# B&R Automation Studio project Lab2_poirts
Automation Studio 4.5.2.102

## Logical view

Binary libraries used (declarations not repeated): Runtime, Operator, AsIecCon, astime, sys_lib, asstring

### Library Logical/Libraries/DriveLib (ANSIC)

#### ConStants.var - Exported constants
```iecst
VAR CONSTANT
	CMD_SWITCHED_ON : USINT := 7;
	CMD_DISABLE_VOLTAGE : USINT := 0;
	CMD_ENABLED : USINT := 15;
	CMD_SHUTDOWN : USINT := 6;
	STATE_READY : USINT := 33;
	STATE_DISABLED : USINT := 64;
	STATE_SWITCHED_ON : USINT := 35;
	ST_INIT : USINT := 0;
	ST_UNKNOWN : USINT := 1;
	ST_OPEN : USINT := 2;
	ST_CLOSE : USINT := 3;
	ST_ACC_POS : USINT := 4;
	ST_ACC_NEG : USINT := 5;
	ST_POS : USINT := 6;
	ST_NEG : USINT := 7;
	ST_DEC_POS : USINT := 8;
	ST_DEC_NEG : USINT := 9;
END_VAR
```

#### DriveLib.fun - Exported functions and function blocks
```iecst
{REDUND_ERROR} FUNCTION_BLOCK DriveStateMachine (*TODO: Add your comment here*) (*$GROUP=User,$CAT=User,$GROUPICON=User.png,$CATICON=User.png*)
	VAR_INPUT
		state : UINT;
		enable : BOOL;
		speed : INT;
	END_VAR
	VAR_OUTPUT
		command : UINT;
	END_VAR
END_FUNCTION_BLOCK

{REDUND_ERROR} FUNCTION_BLOCK DoorStateMachine (*TODO: Add your comment here*) (*$GROUP=User,$CAT=User,$GROUPICON=User.png,$CATICON=User.png*)
	VAR_INPUT
		sw1 : {REDUND_UNREPLICABLE} BOOL;
		sw2 : {REDUND_UNREPLICABLE} BOOL;
		sw3 : {REDUND_UNREPLICABLE} BOOL;
		sw4 : {REDUND_UNREPLICABLE} BOOL;
		direction : {REDUND_UNREPLICABLE} BOOL;
	END_VAR
	VAR_OUTPUT
		speed : {REDUND_UNREPLICABLE} INT;
		state : UINT;
	END_VAR
	VAR
		osw1 : BOOL;
		osw2 : BOOL;
		osw3 : BOOL;
		osw4 : BOOL;
	END_VAR
END_FUNCTION_BLOCK

{REDUND_ERROR} FUNCTION_BLOCK LedStateMachine (*TODO: Add your comment here*) (*$GROUP=User,$CAT=User,$GROUPICON=User.png,$CATICON=User.png*)
	VAR_INPUT
		state : {REDUND_UNREPLICABLE} UINT;
	END_VAR
	VAR_OUTPUT
		led1 : {REDUND_UNREPLICABLE} BOOL;
		led2 : {REDUND_UNREPLICABLE} BOOL;
		led3 : {REDUND_UNREPLICABLE} BOOL;
		led4 : {REDUND_UNREPLICABLE} BOOL;
		timer : {REDUND_UNREPLICABLE} INT := 1;
	END_VAR
END_FUNCTION_BLOCK
```

#### DriveStateMachine.c
```c
#include <bur/plctypes.h>
#ifdef __cplusplus
	extern "C"
	{
#endif
	#include "DriveLib.h"
#ifdef __cplusplus
	};
#endif
/* TODO: Add your comment here */
void DriveStateMachine(struct DriveStateMachine* inst)
{
	UINT mask = inst->state & 0x6f;
	if(!inst->enable)
	{
		inst->command = CMD_SHUTDOWN;
	}
	else
	{
		switch (mask)
		{
			case STATE_DISABLED:
				inst->command = CMD_SHUTDOWN;
				break;

			case STATE_READY:
				inst->command = CMD_ENABLED;
				break;

			case STATE_SWITCHED_ON:
				inst->command = CMD_SWITCHED_ON;
				break;
		}
	}
}
```

#### DoorStateMachine.c
```c
#include <bur/plctypes.h>
#ifdef __cplusplus
	extern "C"
	{
#endif
	#include "DriveLib.h"
#ifdef __cplusplus
	};
#endif
/* TODO: Add your comment here */
void DoorStateMachine(struct DoorStateMachine* inst)
{
	inst->direction=!inst->direction;

	//State init
	/*if(inst->sw1==0 && inst->sw2==0 && inst->sw3==0 && inst->sw4==0)
	{
		inst->state = ST_INIT;
	}
	if(inst->state == ST_INIT)
	{

		inst->state = ST_UNKNOWN;
	}
	//state unknown
	if(inst->state == ST_UNKNOWN)
	{
		inst->state = ST_CLOSE ;
	}*/

	//открытие двери
	if(/*inst->state == ST_CLOSE &&*/ inst->sw1 != inst->osw1 && inst->direction==0)
	{
		inst->state = ST_ACC_POS ;
		inst->speed = -200;
	}

	if(/*inst->state == ST_ACC_POS &&*/ inst->sw2 != inst->osw2 && inst->direction == 0)
	{
		inst->state = ST_POS ;
		inst->speed = -600;
	}

	if(/*inst->state == ST_POS  &&*/ inst->sw3 != inst->osw3 && inst->direction == 0)
	{
		inst->state = ST_DEC_POS;
		inst->speed = -200;
	}

	if(/*inst->state == ST_DEC_POS &&*/ inst->sw4 != inst->osw4 && inst->direction == 0)
	{
		inst->state = ST_OPEN;
		inst->speed = 0;
	}

	//закрытие двери
	if(/*inst->state == ST_OPEN &&*/ inst->sw4 != inst->osw4 && inst->direction==1)
	{
		inst->state = ST_ACC_NEG;
		inst->speed = 200;
	}

	if(/*inst->state == ST_ACC_NEG &&*/ inst->sw3 != inst->osw3 && inst->direction == 1)
	{
		inst->state = ST_NEG;
		inst->speed = 600;
	}

	if(/*inst->state == ST_NEG &&*/ inst->sw2 != inst->osw2 && inst->direction == 1)
	{
		inst->state = ST_DEC_NEG;
		inst->speed = 200;
	}

	if(/*inst->state == ST_DEC_NEG &&*/ inst->sw1 != inst->osw1 && inst->direction == 1)
	{
		inst->state = ST_CLOSE;
		inst->speed = 0;
	}
	inst->osw1 = inst->sw1;
	inst->osw2 = inst->sw2;
	inst->osw3 = inst->sw3;
	inst->osw4 = inst->sw4;

}
```

#### LedStateMachine.c
```c
#include <bur/plctypes.h>
#ifdef __cplusplus
	extern "C"
	{
#endif
	#include "DriveLib.h"
#ifdef __cplusplus
	};
#endif
/* TODO: Add your comment here */
void LedStateMachine(struct LedStateMachine* inst)
{

	if(inst->state == ST_ACC_POS)
	{
		inst->led1 = 0;
		if(inst->timer == 3 )
		{
			inst->led2 = !inst->led2;
		}
		inst->led3 = 1;
		inst->led4 = 1;
	}

	if(inst->state == ST_POS)
	{
		inst->led1 = 0;
		inst->led2 = 0;
		inst->led3 = !inst->led3;
		inst->led4 = 1;
	}

	if(inst->state == ST_DEC_POS)
	{

		inst->led1 = 0;
		inst->led2 = 0;
		inst->led3 = 0;
		if(inst->timer == 3 )
		{
			inst->led4 = !inst->led4;
		}
	}

	if(inst->state == ST_OPEN)
	{
		inst->led1 = 0;
		inst->led2 = 0;
		inst->led3 = 0;
		inst->led4 = 0;
	}

	//закрытие двери
	if(inst->state == ST_ACC_NEG )
	{
		inst->led1 = 0;
		inst->led2 = 0;
		if(inst->timer == 3 )
		{
			inst->led3 = !inst->led3;
		}
		inst->led4 = 1;
	}

	if(inst->state == ST_NEG)
	{
		inst->led1 = 0;
		inst->led2 =!inst->led2;
		inst->led3 = 1;
		inst->led4 = 1;
	}

	if(inst->state == ST_DEC_NEG )
	{
		if(inst->timer == 3 )
		{
			inst->led1 = !inst->led1;
		}
		inst->led2 = 1;
		inst->led3 = 1;
		inst->led4 = 1;
	}

	if(inst->state == ST_CLOSE)
	{
		inst->led1 = 1;
		inst->led2 = 1;
		inst->led3 = 1;
		inst->led4 = 1;
	}

	if(inst->timer == 3)
		inst->timer = 0;

	inst->timer++;
}
```

### Program Logical/Program (ANSIC)

#### Init.c - Initialization code
```c
#include <bur/plctypes.h>

#ifdef _DEFAULT_INCLUDES
	#include <AsDefault.h>
#endif

void _INIT ProgramInit(void)
{

	DriveSM.enable = 1;
}
```

#### Cyclic.c - Cyclic code
```c
#include <bur/plctypes.h>

#ifdef _DEFAULT_INCLUDES
	#include <AsDefault.h>
#endif

void _CYCLIC ProgramCyclic(void)
{
	DoorStateMachine(&DoorSM);
	DriveSM.speed = DoorSM.speed;
	DriveStateMachine(&DriveSM);
	LedSM.state = DoorSM.state;
	LedStateMachine(&LedSM);
	/*
	DriveSM.speed = 250;
	DriveStateMachine(&DriveSM);
*/
}
```

#### Variables.var - Local variables
```iecst
VAR
	speed : INT := 0;
	DriveSM : DriveStateMachine := (0);
	LedSM : LedStateMachine := (0);
	DoorSM : DoorStateMachine := (0);
END_VAR
```

Listed in the project but not available here: Logical/Libraries/DriveLib/Types.typ, Logical/Program/Exit.c, Logical/Program/Types.typ
